Staubli VAL3: KIT.pjx

--- KIT.pjx ---
Parameters version=s7.7 stackSize=5000 millimeterUnit=true
Program file=Align.pgx
Program file=ExtraSysAxisIni.pgx
Program file=GoHome.pgx
Program file=Poll.pgx
Program file=RecordAlarm.pgx
Program file=start.pgx
Program file=stop.pgx
Program file=TrajByPass.pgx
Program file=UpLoad.pgx
Data file=Kit.dtx
Library alias=UI path=Disk://StaubliUI/StaubliUI.pjx
Library alias=TxtFile path=Disk://TxtFile/TxtFile.pjx
Library alias=DataBase path=Disk://DataBase/DataBase.pjx
Library alias=IO path=Disk://IO/IO.pjx
Library alias=ExtAxis path=Disk://extAxisCan/extAxisCan.pjx autoload=false
Library alias=Custom path=Disk://Custom/Custom.pjx

--- KIT.dtx ---
mdesc mNomSpeed
bool bSync
num nFileID

--- ALIGN.pgx ---
public program Align(tool x_tTool)
  local point l_pPoint
  local num l_nKey
  local bool l_bRes
begin
  //-----------------------------------------------------------------------
  //Header begin
  //Description of program
  //  工具对齐
  //Input parameters
  //  tool x_TxtFile:tCfg:工具值
  //Output paramaters
  //  bool x_bOK:是否对齐
  //Example
  //  call Align(tool,bOK)
  //History
  //  Creation : 2012-06-11 - PF.Zhong
  //Header end
  //不推荐客户自己改动此函数代码
  //-----------------------------------------------------------------------
  resetMotion()
  cls()
  link(l_pPoint,world)
  l_pPoint=here(TxtFile:tCfg,world)
  l_pPoint.trsf=align(l_pPoint.trsf,world.trsf)
  mNomSpeed.blend=off
  movej(l_pPoint,TxtFile:tCfg,mNomSpeed)
  call UI:Control_PanelMd("正在对齐,请稍候")
  call UI:Control_BottomS(",,,,,,,终止")
  while !isEmpty()
    l_nKey=getKey()
    switch l_nKey
      case 278
        call UI:Control_YesNO("确定需要终止吗?",l_bRes)
        cls()
        if l_bRes
          resetMotion()
          return
        else
          call UI:Control_PanelMd("正在对齐,请稍候")
          call UI:Control_BottomS(",,,,,,,终止")
        endIf

      break

    endSwitch
    delay(0)
  endWhile
  cls()
  call UI:Control_PanelMd("对齐成功!")
  delay(2)
  cls()
  delay(0)
end

--- ExtraSysAxisIni.pgx ---
public program ExtraSysAxisIni(bool& x_bRes)
begin

  //2014.07.28
  //同步七八轴

  x_bRes=false
  TxtFile:bSync7Axis=TxtFile:bSync8Axis=false
  if $fileExists("Usr://configs/externaxes.cfx") and getVersion("externalAxis")!="false"

    if !ExtAxis:libExist("Disk://extAxisCan/extAxisCan.pjx")

      //2014.08.06
      //适配7.5版本和S7.6版本
      if find(getVersion("System"),"s7.5")>=0
        if !$copy("Disk://extAxisCan/TASK4MS7.5.pgx","Disk://extAxisCan/TASK4MS.pgx")
          popUpMsg("外部轴TASK4MS程序不正确")
          return
        endIf

      else
        if !$copy("Disk://extAxisCan/TASK4MS7.6.pgx","Disk://extAxisCan/TASK4MS.pgx")
          popUpMsg("外部轴TASK4MS程序不正确")
          return
        endIf
      endIf

      //


      if ExtAxis:libLoad("Disk://extAxisCan/extAxisCan.pjx")!=0
        popUpMsg("加载同步轴库不正确")
        return
      endIf
    endIf
    call ExtAxis:CheckAxis(TxtFile:bSync7Axis,TxtFile:bSync8Axis)
    call ExtAxis:init()
    // call ExtAxis:Reset()
    DataBase:nAsysAxisPer=max(0.004,DataBase:nAsysAxisPer)
    taskCreateSync "SyncAxis",DataBase:nAsysAxisPer,bSync,ExtAxis:Task4ms()

  endIf

  x_bRes=true





end

--- GOHOME.pgx ---
public program GoHome()
  local num l_nKey
  local bool l_bRes
  local trsf l_trTrsf
  local point l_p
begin
  //机械手臂回零程序


  //2014.07.28
  //同步七八轴
//  if TxtFile:bSync7Axis or TxtFile:bSync8Axis
//    if !ExtAxis:libExist("Disk://extAxisCan/extAxisCan.pjx")
//      if ExtAxis:libLoad("Disk://extAxisCan/extAxisCan.pjx")!=0
//        popUpMsg("加载外部轴出错")
//        return
//      endIf
//    endIf
//  endIf

  //回零程序
  cls()
  resetMotion()
  call UI:Form_MainS(",,,,,,,终止")
  call UI:Control_PanelMd("机器人正在回零")
  DataBase:mJHome.tvel=min(500,max(50,TxtFile:nHomeSpeed*1000/60))
  DataBase:mJHome.blend=off


  //2014.07.29 同步七轴或者八轴
  if TxtFile:bSync7Axis or TxtFile:bSync8Axis
    l_trTrsf.x=TxtFile:trSync7Axis.y
    l_trTrsf.y=TxtFile:trSync8Axis.y
    call ExtAxis:SingleMove(1,TxtFile:jHome,l_p,l_p,TxtFile:tCfg,DataBase:mJHome,l_trTrsf)
  else
    movej(TxtFile:jHome,TxtFile:tCfg,DataBase:mJHome)

  endIf

  wait(!isEmpty()and getKey()==-1)
  while  !isEmpty()
    l_nKey=getKey()
    switch l_nKey
      case 278
        call UI:Control_YesNO("确定要终止回零吗?",l_bRes)
        if l_bRes
          resetMotion()
          return
        else
          call UI:Form_MainS(",,,,,,,终止")
          call UI:Control_PanelMd("机器人正在回零")
        endIf
      break
    endSwitch
    delay(0)
  endWhile
  wait(DataBase:bIsHome)


  //2014.12.09
  //外部PLC控制回零信号
  if DataBase:bExtraContrAxis

    call IO:AtHomePulse()

  endIf
  //************************



  cls()
  call UI:Control_PanelMd("回零成功")
  delay(2)
  cls()
end

--- POLL.pgx ---
public program Poll()
  local num l_nNum
  local num l_nBuffTime
  local bool l_bIsAlarm
begin
    //不推荐客户自己改动此函数代码
  //-----------------------------------------------------------------------
  //轮询
  //MoveID
  DataBase:nID=getMoveId()
  DataBase:jCurrentJoint=herej()
  DataBase:pCurrentPoint=here(TxtFile:tCfg,world)
  l_nNum=abs(DataBase:jCurrentJoint.j1-TxtFile:jHome.j1)+abs(DataBase:jCurrentJoint.j2-TxtFile:jHome.j2)+abs(DataBase:jCurrentJoint.j3-TxtFile:jHome.j3)
  l_nNum= l_nNum+abs(DataBase:jCurrentJoint.j4-TxtFile:jHome.j4)+abs(DataBase:jCurrentJoint.j5-TxtFile:jHome.j5)+abs(DataBase:jCurrentJoint.j6-TxtFile:jHome.j6)
  DataBase:bIsHome=l_nNum<0.3


  //实时轮询
  while  true

    //一般在读写文本的时候，对bStopPoll停止

    //2016.03.24
    //为天其
    if esStatus()==2
      if l_bIsAlarm==false
        l_bIsAlarm=true
        call RecordAlarm()
      endIf
    else
      l_bIsAlarm=false
    endIf
    //**************


    //模式
    l_nBuffTime=clock()
    call IO:Alarm(TxtFile:trIODelay.ry,DataBase:nInterfaceType,DataBase:bAlarm)
    if !DataBase:bStopPoll
      //查看是否上电
      DataBase:nToolMode=workingMode()
      DataBase:bPowerOn=isPowered()
      call IO:GetPreset(DataBase:nPresetData,TxtFile:trPresetData.z,TxtFile:trPresetData.x,TxtFile:trPresetData.y)
      //掉点以后，安全IO
      if !DataBase:bPowerOn
        call IO:SafteyIO()
        DataBase:bAirOn=DataBase:bFollowOn=DataBase:bLaserOn=false
        //   DataBase:nPresetData[0]=DataBase:nPresetData[1]=DataBase:nPresetData[2]=DataBase:nPresetData[3]=DataBase:nPresetData[4]=0
      else

        call IO:GetKeyIO(DataBase:bAirOn,DataBase:bFollowOn,DataBase:bLaserOn)

        //机器人实时线速度
        DataBase:nRobotSpeed=getSpeed(TxtFile:tCfg)

        //2014.3.24 设置机器人速度到O2_aNull
        call IO:SendSpeed(DataBase:nRobotSpeed)
        //MoveID
        DataBase:nID=getMoveId()

        //机器人位置
        DataBase:jCurrentJoint=herej()
        DataBase:pCurrentPoint=here(TxtFile:tCfg,world)

        //检查是否在Home
        //        l_nNum=abs(DataBase:jCurrentJoint.j1-TxtFile:jHome.j1)+abs(DataBase:jCurrentJoint.j2-TxtFile:jHome.j2)+abs(DataBase:jCurrentJoint.j3-TxtFile:jHome.j3)
        //        l_nNum= l_nNum+abs(DataBase:jCurrentJoint.j4-TxtFile:jHome.j4)+abs(DataBase:jCurrentJoint.j5-TxtFile:jHome.j5)+abs(DataBase:jCurrentJoint.j6-TxtFile:jHome.j6)
        //        DataBase:bIsHome=l_nNum<0.1

        //代码重构
        DataBase:bIsHome=distance(jointToPoint(flange,world,DataBase:jCurrentJoint),jointToPoint(flange,world,TxtFile:jHome))<0.1

      endIf



      //用户自定义轮询
      call Custom:CustomPoll()

      //数字量转换为模拟量
      if  DataBase:nPointType==0 or !TxtFile:bWeldEnable  or !DataBase:bMoveTask
        call IO:Digtal2Analog()
      endIf
    endIf


    //2014.12.11
    //*************************
    if TxtFile:bSync7Axis or TxtFile:bSync8Axis
     if taskStatus("SyncAxis")!=1 and DataBase:bPowerOn

      disablePower()
    endIf

    //*******************
    endIf




    delay(0)

    //每次poll循环需要的时间
    DataBase:nPollTime=clock()-l_nBuffTime
  endWhile


end

--- RecordAlarm.pgx ---
program RecordAlarm()
  local string l_sString
  local joint l_jJoint
begin
  if !$fileExists("Log://alarm.txt")
    nFileID=$fileOpen("Log://alarm.txt","w")
  else
    nFileID=$fileOpen("Log://alarm.txt","a")
  endIf



  if nFileID<0 or nFileID>9
    return
  endIf

  l_sString=getDate("%Y_%m_%d %H:%M:%S")
  l_sString=l_sString+"急停触发:产品:"+DataBase:sProductName[DataBase:nWorkPlaceIndex]+"路径:"+toString("",DataBase:nTrajIndex)
  l_sString=l_sString+"MoveID:"+toString(".3",getMoveId())

  $fileSet(nFileID,l_sString,1)
  l_jJoint=herej()

  l_sString="关节位置:"+toString(".3",l_jJoint.j1)+","+toString(".3",l_jJoint.j2)+","+toString(".3",l_jJoint.j3)+","
  l_sString= l_sString+toString(".3",l_jJoint.j4)+","+toString(".3",l_jJoint.j5)+","+toString(".3",l_jJoint.j6)

   $fileSet(nFileID,l_sString,1)

   $fileClose(nFileID)









end

--- TrajByPass.pgx ---
public program TrajByPass(num x_nIndex, num x_nTotal)
begin


 // 路径由外部信号过滤
 // 实现方式
 //通过一个数字量输入信号，一个模拟量输入信号，一个模拟量输出信号
 //没有经过测试过



  do

    call IO:TrajBypass(TxtFile:bBypass[x_nIndex-1],x_nIndex-1)
    x_nIndex=x_nIndex+1
    delay(0)
  until TxtFile:bBypass[x_nIndex-1]==false or x_nIndex>=x_nTotal



end

--- UPLOAD.pgx ---
public program UpLoad()
  local num l_nKey
  local bool l_bRes
  local num l_nTime
begin
  //不推荐客户自己改动此函数代码
  //-----------------------------------------------------------------------
  //把CS8C的信息上传到上位机中
  cls()
  call UI:Control_PanelMd("正在上传，请等待")
  call UI:Control_BottomS(",,,,,,,终止")
  call TxtFile:CloseFile()
  DataBase:bUpload=true
  l_nTime=clock()


  //开始上传
  while DataBase:bUpload==true and 120-clock()+l_nTime>0
    l_nKey=getKey()

    if l_nKey==278
      call UI:Control_YesNO("确定要终止上传吗",l_bRes)
      if l_bRes
        DataBase:bUpload=false
        return
      else
        call UI:Control_PanelMd("正在上传，请等待")
        call UI:Control_BottomS(",,,,,,,终止")
      endIf
    endIf


    gotoxy(0,12)
    put("剩余:"+toString("",120-clock()+l_nTime)+"秒     ")
    delay(0)

  endWhile

  //对上传结果进行判断
  DataBase:bUpload=false
  if clock()>l_nTime+60
    popUpMsg("上传失败!")
  else
    popUpMsg("上传成功")
  endIf
  cls()

end
